// TIA Portal V21 export
TYPE "coneCrusherInterface"
   STRUCT
      cmd { ExternalAccessible := 'False'; ExternalVisible := 'False'; ExternalWritable := 'False'} : "coneCrusherCmd";
      sta { ExternalAccessible := 'False'; ExternalVisible := 'False'; ExternalWritable := 'False'; S7_SetPoint := 'True'} : "coneCrusherSta";
      out { ExternalAccessible := 'False'; ExternalVisible := 'False'; ExternalWritable := 'False'; S7_SetPoint := 'True'} : "coneCrusherOut";
   END_STRUCT;
END_TYPE
